ABB RAPID module: Module1.mod

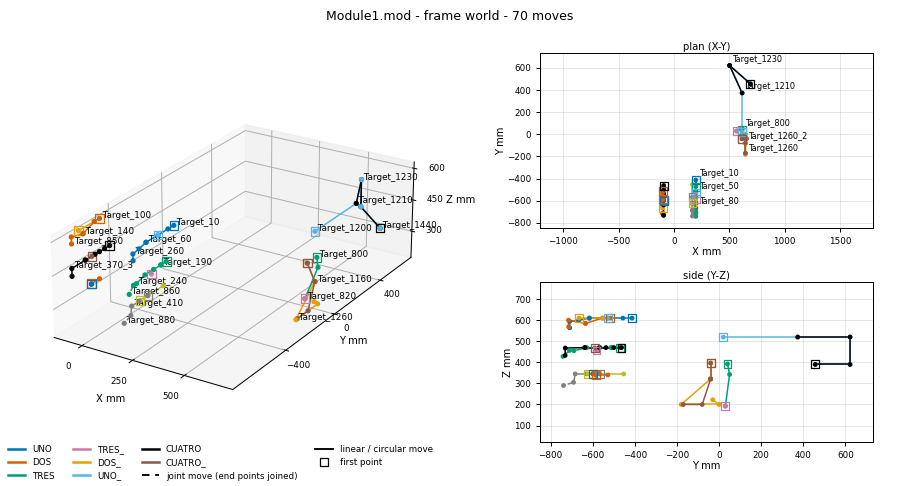
[picture p0: tool path of Module1.mod in frame world, 70 of 71 moves have a stored position in this frame; points joined in program order, loops and branches not executed]
MODULE Module1
    CONST robtarget Target_10:=[[445,309.451,360],[0,0.707106781,0.707106781,0],[-1,0,0,0],[9E+09,9E+09,9E+09,9E+09,9E+09,9E+09]];
    CONST robtarget Target_30:=[[445.000100716,265.84797315,360.000005505],[0.204070481,0.677019397,0.677019332,-0.204070573],[-1,-1,0,0],[9E+09,9E+09,9E+09,9E+09,9E+09,9E+09]];
    CONST robtarget Target_50:=[[444.999989498,193.403179869,359.99999842],[0.39678617,0.585286862,0.58528689,-0.396786191],[-1,-2,1,0],[9E+09,9E+09,9E+09,9E+09,9E+09,9E+09]];
    CONST robtarget Target_60:=[[445.000001173,106.761011861,360.000002181],[0.396786171,0.585286826,0.585286919,-0.3967862],[-1,-2,1,0],[9E+09,9E+09,9E+09,9E+09,9E+09,9E+09]];
    CONST robtarget Target_70:=[[444.999995441,106.761019962,359.999988422],[0.498060694,0.501931741,0.501931802,-0.498060778],[-1,-2,1,0],[9E+09,9E+09,9E+09,9E+09,9E+09,9E+09]];
    CONST robtarget Target_80:=[[445,56.559774308,350],[0.498058869,0.50193349,0.501933625,-0.498059004],[-1,-2,1,0],[9E+09,9E+09,9E+09,9E+09,9E+09,9E+09]];
    CONST robtarget Target_260:=[[445,13.051774308,344.078],[0.498058632,0.501933253,0.501933862,-0.498059241],[-1,-2,1,0],[9E+09,9E+09,9E+09,9E+09,9E+09,9E+09]];
    CONST robtarget Target_840:=[[445,13.283774308,314.079],[0.498058666,0.501933287,0.501933828,-0.498059207],[-1,-2,1,0],[9E+09,9E+09,9E+09,9E+09,9E+09,9E+09]];
    CONST robtarget Target_100:=[[145,206.823,360],[0,0.707106781,0.707106781,0],[-2,0,-1,0],[9E+09,9E+09,9E+09,9E+09,9E+09,9E+09]];
    CONST robtarget Target_120:=[[145.000023763,169.277992134,359.999994736],[0.208753422,0.675590111,0.675590131,-0.208753407],[-2,0,-1,0],[9E+09,9E+09,9E+09,9E+09,9E+09,9E+09]];
    CONST robtarget Target_140:=[[145,89.022774308,335],[0.308604589,0.636210034,0.636210034,-0.308604589],[-2,0,-1,0],[9E+09,9E+09,9E+09,9E+09,9E+09,9E+09]];
    CONST robtarget Target_150:=[[145,87.832774308,335],[0.308604589,0.636210034,0.636210034,-0.308604589],[-2,0,-1,0],[9E+09,9E+09,9E+09,9E+09,9E+09,9E+09]];
    CONST robtarget Target_160:=[[145,7.662774308,350.108],[0.495529584,0.504430646,0.504430801,-0.495529739],[-2,1,-2,0],[9E+09,9E+09,9E+09,9E+09,9E+09,9E+09]];
    CONST robtarget Target_850:=[[145,8.374774308,319.114],[0.495529584,0.504430646,0.504430801,-0.495529739],[-2,1,-2,0],[9E+09,9E+09,9E+09,9E+09,9E+09,9E+09]];
    CONST robtarget Target_180:=[[445,250.207,220],[0,0.707106781,0.707106781,0],[0,0,0,0],[9E+09,9E+09,9E+09,9E+09,9E+09,9E+09]];
    CONST robtarget Target_190:=[[445,210.045,220],[0,0.707106781,0.707106781,0],[-1,0,0,0],[9E+09,9E+09,9E+09,9E+09,9E+09,9E+09]];
    CONST robtarget Target_210:=[[444.999974423,210.04498181,219.999975641],[0.196714093,0.67919333,0.679193304,-0.196714112],[-1,-1,1,0],[9E+09,9E+09,9E+09,9E+09,9E+09,9E+09]];
    CONST robtarget Target_220:=[[444.999969721,157.562432775,220.000153936],[0.196714096,0.679193328,0.679193306,-0.196714111],[-1,-1,0,0],[9E+09,9E+09,9E+09,9E+09,9E+09,9E+09]];
    CONST robtarget Target_230:=[[445.000020297,94.798793532,219.999986793],[0.490571323,0.509254076,0.509254286,-0.490571233],[-1,-2,1,0],[9E+09,9E+09,9E+09,9E+09,9E+09,9E+09]];
    CONST robtarget Target_240:=[[444.99998259,33.260372465,205.010464734],[0.490571277,0.509254086,0.509254311,-0.490571243],[-1,-2,1,0],[9E+09,9E+09,9E+09,9E+09,9E+09,9E+09]];
    CONST robtarget Target_300:=[[445,12.043774308,205.998],[0.490571564,0.509254226,0.5092539,-0.490571238],[-1,-2,1,0],[9E+09,9E+09,9E+09,9E+09,9E+09,9E+09]];
    CONST robtarget Target_860:=[[445,-18.461225692,178.026],[0.49056712,0.509258507,0.509249619,-0.490575682],[-1,-2,1,0],[9E+09,9E+09,9E+09,9E+09,9E+09,9E+09]];
    CONST robtarget Target_300_2:=[[445.000076449,140.791521426,205.991567014],[0.490571145,0.509254485,0.509253958,-0.490571328],[-1,-2,1,0],[9E+09,9E+09,9E+09,9E+09,9E+09,9E+09]];
    CONST robtarget Target_170:=[[145.000002632,57.832569204,360.00000345],[0.49552756,0.504432594,0.504432809,-0.495527736],[-2,1,-2,0],[9E+09,9E+09,9E+09,9E+09,9E+09,9E+09]];
    CONST robtarget Target_120_2:=[[145.000023763,169.277992134,359.999994736],[0.208753422,0.675590111,0.675590131,-0.208753407],[-2,0,-1,0],[9E+09,9E+09,9E+09,9E+09,9E+09,9E+09]];
    CONST robtarget Target_50_2:=[[444.999989498,193.403179869,359.99999842],[0.39678617,0.585286862,0.58528689,-0.396786191],[-1,-2,1,0],[9E+09,9E+09,9E+09,9E+09,9E+09,9E+09]];
    CONST jointtarget hoome:=[[0,0,0,0,30,0],[9E+09,9E+09,9E+09,9E+09,9E+09,9E+09]];
    CONST robtarget Target_310:=[[155,259.373,220],[0,0.707106781,0.707106781,0],[-2,0,-1,0],[9E+09,9E+09,9E+09,9E+09,9E+09,9E+09]];
    CONST robtarget Target_320:=[[155,222.546,220],[0,0.707106781,0.707106781,0],[-2,0,-1,0],[9E+09,9E+09,9E+09,9E+09,9E+09,9E+09]];
    CONST robtarget Target_330:=[[154.999993427,185.47297748,219.999991899],[0.181722193,0.68335719,0.683357178,-0.181722213],[-2,0,-1,0],[9E+09,9E+09,9E+09,9E+09,9E+09,9E+09]];
    CONST robtarget Target_340:=[[155,153.836774308,220],[0.181724929,0.683356459,0.683356459,-0.181724929],[-2,0,-1,0],[9E+09,9E+09,9E+09,9E+09,9E+09,9E+09]];
    CONST robtarget Target_350:=[[155.000000465,85.426287942,219.999986272],[0.351807406,0.613377267,0.613377023,-0.351807484],[-2,1,-2,0],[9E+09,9E+09,9E+09,9E+09,9E+09,9E+09]];
    CONST robtarget Target_360:=[[155.000020231,85.426284038,219.999972166],[0.502982262,0.496999972,0.496999701,-0.502982276],[-2,1,-2,0],[9E+09,9E+09,9E+09,9E+09,9E+09,9E+09]];
    CONST robtarget Target_370_3:=[[154.117650914,-7.63964163,217.880472499],[0.502982249,0.496999966,0.496999703,-0.502982293],[-2,1,-2,0],[9E+09,9E+09,9E+09,9E+09,9E+09,9E+09]];
    CONST robtarget Target_870:=[[154.117692068,-8.05845949,182.882972826],[0.502982281,0.497000006,0.496999676,-0.502982246],[-2,1,-2,0],[9E+09,9E+09,9E+09,9E+09,9E+09,9E+09]];
    CONST robtarget Target_370_2:=[[154.117693643,132.374266615,218.205277098],[0.502982249,0.496999966,0.496999703,-0.502982293],[-2,1,-2,0],[9E+09,9E+09,9E+09,9E+09,9E+09,9E+09]];
    CONST robtarget Target_390:=[[415.000021736,155.814134714,94.99994956],[0.222483326,0.671193787,0.671193888,-0.222483337],[-1,-2,1,0],[9E+09,9E+09,9E+09,9E+09,9E+09,9E+09]];
    CONST robtarget Target_400:=[[414.999964418,93.028686316,95.000070499],[0.494470801,0.505469141,0.505468247,-0.494470854],[-1,-2,1,0],[9E+09,9E+09,9E+09,9E+09,9E+09,9E+09]];
    CONST robtarget Target_410:=[[414.999780299,39.624514396,95.000017901],[0.494470475,0.505469266,0.505467893,-0.494471414],[-1,-2,1,0],[9E+09,9E+09,9E+09,9E+09,9E+09,9E+09]];
    CONST robtarget Target_420_2:=[[415,31.615774308,55.006],[0.49447229,0.505467643,0.505467259,-0.494471906],[-1,-2,1,0],[9E+09,9E+09,9E+09,9E+09,9E+09,9E+09]];
    CONST robtarget Target_880:=[[415.000153001,-15.724115102,40.013288948],[0.49447062,0.505469365,0.505467764,-0.4944713],[-1,-2,1,0],[9E+09,9E+09,9E+09,9E+09,9E+09,9E+09]];
    CONST robtarget Target_430:=[[415.000047641,100.795599035,94.999989609],[0.494470604,0.505469297,0.505467834,-0.494471315],[-1,-2,1,0],[9E+09,9E+09,9E+09,9E+09,9E+09,9E+09]];
    CONST robtarget Target_380:=[[415,269.946,95],[0,0.707106781,0.707106781,0],[-1,0,0,0],[9E+09,9E+09,9E+09,9E+09,9E+09,9E+09]];
    CONST robtarget Target_910:=[[154.999998327,259.37294151,90.000018028],[-0.000000019,0.707106797,0.707106766,-0.000000028],[-2,0,-1,0],[9E+09,9E+09,9E+09,9E+09,9E+09,9E+09]];
    CONST robtarget Target_930:=[[155.000007698,111.881805431,90.000010525],[0.506551604,0.493361374,0.493361398,-0.506551635],[-2,1,-2,0],[9E+09,9E+09,9E+09,9E+09,9E+09,9E+09]];
    CONST robtarget Target_940:=[[155.00014811,-18.072997939,93.429168302],[0.506551657,0.493361261,0.493361508,-0.506551583],[-2,1,-2,0],[9E+09,9E+09,9E+09,9E+09,9E+09,9E+09]];
    CONST robtarget Target_950:=[[155.000223386,-19.39194722,43.446578802],[0.506551723,0.493361207,0.493361565,-0.506551516],[-2,1,-2,0],[9E+09,9E+09,9E+09,9E+09,9E+09,9E+09]];
    CONST robtarget Target_480:=[[144.999909688,137.135818312,89.9999693],[0.497141997,0.502841197,0.502842112,-0.497142208],[-2,1,-2,0],[9E+09,9E+09,9E+09,9E+09,9E+09,9E+09]];
    CONST robtarget Target_470:=[[144.999992416,137.13583322,89.999952579],[0.158251404,0.689170827,0.689170921,-0.1582514],[-2,0,-1,0],[9E+09,9E+09,9E+09,9E+09,9E+09,9E+09]];
    CONST robtarget Target_460:=[[145,194.615,90],[0,0.707106781,0.707106781,0],[-2,0,-1,0],[9E+09,9E+09,9E+09,9E+09,9E+09,9E+09]];
    CONST robtarget Target_800:=[[15.000003085,20,-7.279986715],[0.001374548,-0.707105336,0.707105556,-0.001373609],[0,-1,-1,0],[9E+09,9E+09,9E+09,9E+09,9E+09,9E+09]];
    CONST robtarget Target_810:=[[15.194319396,30.000063266,-57.279608845],[0.001374525,-0.707105304,0.707105589,-0.001373591],[0,-1,-1,0],[9E+09,9E+09,9E+09,9E+09,9E+09,9E+09]];
    CONST robtarget Target_820:=[[-34.3,9.999774308,-207.473],[0.001376059,-0.707105442,0.707105442,-0.001376059],[0,-1,-1,0],[9E+09,9E+09,9E+09,9E+09,9E+09,9E+09]];
    CONST robtarget Target_830:=[[16.049330824,30.000353686,-277.277947373],[0.001374525,-0.707105304,0.707105589,-0.001373591],[0,-1,-1,0],[9E+09,9E+09,9E+09,9E+09,9E+09,9E+09]];
    CONST robtarget Target_960:=[[15,-60.000225692,-3.34],[0.422618262,0,0.906307787,0],[-1,0,-1,0],[9E+09,9E+09,9E+09,9E+09,9E+09,9E+09]];
    CONST robtarget Target_980:=[[15.000003989,-60.000225846,-65.005610701],[0.698090332,-0.000000037,0.716009699,-0.000000028],[-1,1,-2,0],[9E+09,9E+09,9E+09,9E+09,9E+09,9E+09]];
    CONST robtarget Target_990:=[[64.983949086,-84.888859881,-188.758694739],[0.698090343,-0.000000088,0.716009688,0.00000008],[-1,1,-2,0],[9E+09,9E+09,9E+09,9E+09,9E+09,9E+09]];
    CONST robtarget Target_1000:=[[64.983940199,-84.888856272,-260.223415545],[0.698090318,-0.000000083,0.716009712,0.000000092],[-1,1,-2,0],[9E+09,9E+09,9E+09,9E+09,9E+09,9E+09]];
    CONST robtarget Target_1010:=[[64.983925895,-54.888697083,-260.223308264],[0.698090428,-0.000000715,0.716009604,0.000000241],[-1,1,-2,0],[9E+09,9E+09,9E+09,9E+09,9E+09,9E+09]];
    CONST robtarget Target_1020:=[[67.517875393,-54.888638408,-160.255409875],[0.698090412,-0.000000696,0.716009621,0.000000195],[-1,1,-2,0],[9E+09,9E+09,9E+09,9E+09,9E+09,9E+09]];
    CONST robtarget Target_1030:=[[1115.000003258,-650.827226308,222.202998223],[0.342020143,0,0.939692621,0],[0,-1,0,0],[9E+09,9E+09,9E+09,9E+09,9E+09,9E+09]];
    CONST robtarget Target_1040:=[[1115.000009669,-650.827230544,392.898398622],[0.683149215,-0.147345411,0.700684713,0.143657274],[-1,1,-2,0],[9E+09,9E+09,9E+09,9E+09,9E+09,9E+09]];
    CONST robtarget Target_1050:=[[1115.000011784,-558.507726654,392.898390868],[0.683149204,-0.14734549,0.700684704,0.143657288],[0,1,-2,0],[9E+09,9E+09,9E+09,9E+09,9E+09,9E+09]];
    CONST robtarget Target_1060:=[[1115.000006212,-451.354920054,392.898384166],[0.683149189,-0.14734552,0.700684714,0.143657286],[0,1,-2,0],[9E+09,9E+09,9E+09,9E+09,9E+09,9E+09]];
    CONST robtarget Target_1080:=[[998.889389949,-391.005407979,392.898398132],[0.683149203,-0.147345556,0.700684696,0.143657271],[0,2,-3,0],[9E+09,9E+09,9E+09,9E+09,9E+09,9E+09]];
    CONST robtarget Target_1090:=[[865.105301275,-168.564929633,392.898396083],[0.616538883,-0.335834912,0.632364278,0.327429593],[0,1,-2,0],[9E+09,9E+09,9E+09,9E+09,9E+09,9E+09]];
    CONST robtarget Target_1100:=[[878.271514464,-30.097814532,392.898393764],[0.616538885,-0.335835049,0.632364231,0.327429538],[0,2,-3,0],[9E+09,9E+09,9E+09,9E+09,9E+09,9E+09]];
    CONST robtarget Target_1110:=[[878.271453157,-30.097779623,331.594271959],[0.616538889,-0.33583503,0.632364227,0.327429558],[0,2,-3,0],[9E+09,9E+09,9E+09,9E+09,9E+09,9E+09]];
    CONST robtarget Target_1120:=[[927.980685621,-63.698381666,331.594348136],[0.6165389,-0.335835004,0.632364219,0.32742958],[0,1,-2,0],[9E+09,9E+09,9E+09,9E+09,9E+09,9E+09]];
    CONST robtarget Target_1130:=[[929.115831572,-62.018793499,411.568574487],[0.616538876,-0.335835031,0.63236422,0.327429593],[0,1,-2,0],[9E+09,9E+09,9E+09,9E+09,9E+09,9E+09]];
    CONST robtarget Target_1140:=[[155.00004953,123.02170152,95.65965675],[0.494470878,0.50546913,0.505468146,-0.494470891],[-2,1,-2,0],[9E+09,9E+09,9E+09,9E+09,9E+09,9E+09]];
    CONST robtarget Target_1190:=[[45,-50.000225692,-177.596],[0.574790179,-0.270574227,0.743396577,-0.209206516],[-1,0,-1,0],[9E+09,9E+09,9E+09,9E+09,9E+09,9E+09]];
    CONST robtarget Target_1170:=[[15,-100.000225692,-269.732],[0.342020143,0,0.939692621,0],[-1,0,-1,0],[9E+09,9E+09,9E+09,9E+09,9E+09,9E+09]];
    CONST robtarget Target_1180:=[[45,-50.000225692,-271.262],[0.611678933,0,0.791106114,0],[-1,0,-1,0],[9E+09,9E+09,9E+09,9E+09,9E+09,9E+09]];
    CONST robtarget Target_1260:=[[45,-200.000225692,-200],[0.602385883,-0.137375677,0.779087162,-0.106218474],[-1,1,-2,0],[9E+09,9E+09,9E+09,9E+09,9E+09,9E+09]];
    CONST robtarget Target_1150:=[[15,-60.000225692,-24.284],[0.173648178,0,0.984807753,0],[-1,0,-1,0],[9E+09,9E+09,9E+09,9E+09,9E+09,9E+09]];
    CONST robtarget Target_1160:=[[52.587704822,-60.000225692,-78.767194242],[0.173648178,0,0.984807753,0],[-1,0,-1,0],[9E+09,9E+09,9E+09,9E+09,9E+09,9E+09]];
    CONST robtarget Target_1250:=[[1167.584,-194.402225692,410],[0.31160272,-0.387399417,0.856121436,0.141001857],[0,0,-1,0],[9E+09,9E+09,9E+09,9E+09,9E+09,9E+09]];
    CONST robtarget Target_1240:=[[1002.320747823,-49.18417527,390.000000069],[0.341036269,-0.656847149,0.671992582,0.025924035],[0,0,-1,0],[9E+09,9E+09,9E+09,9E+09,9E+09,9E+09]];
    CONST robtarget Target_1230:=[[1002.32107139,-49.183439733,519.999883014],[0.311602972,-0.387398085,0.856122024,0.141001388],[0,0,-1,0],[9E+09,9E+09,9E+09,9E+09,9E+09,9E+09]];
    CONST robtarget Target_1210:=[[1115.000004816,-297.587934649,519.999950749],[0.342020175,0.00000003,0.939692609,-0.000000022],[0,-1,0,0],[9E+09,9E+09,9E+09,9E+09,9E+09,9E+09]];
    CONST robtarget Target_1200:=[[1115,-650.827225692,520],[0.342020143,0,0.939692621,0],[0,-1,0,0],[9E+09,9E+09,9E+09,9E+09,9E+09,9E+09]];
    CONST robtarget Target_1280:=[[52.587712308,-60.000227715,-78.767220897],[0.440689623,-0.000000022,0.897659543,-0.000000013],[-1,0,-1,0],[9E+09,9E+09,9E+09,9E+09,9E+09,9E+09]];
    CONST robtarget Target_1440:=[[1190.119504813,-214.204262911,389.999988496],[0.341036269,-0.656847149,0.671992582,0.025924035],[0,0,-1,0],[9E+09,9E+09,9E+09,9E+09,9E+09,9E+09]];
    CONST robtarget Target_1260_2:=[[45,-100.000225692,-200],[0.554368788,-0.334338154,0.716984512,-0.258508131],[-1,1,-2,0],[9E+09,9E+09,9E+09,9E+09,9E+09,9E+09]];
    CONST robtarget Target_1460:=[[45.000159369,-190.000214557,-199.999516221],[0.611679058,-0.000002498,0.791106017,-0.000001528],[-1,1,-2,0],[9E+09,9E+09,9E+09,9E+09,9E+09,9E+09]];

PROC main()
    WaitDI DI_01,1;  // Espera hasta que la entrada DI_01 sea igual a 1.
    SETDO DO_03,1;   // Establece la salida DO_03 en 1.
    homee;           // Mueve el robot a la posición de origen (home).
    BaldeR;          // Toma el balde de la banda.
    homee;           // Vuelve a la posición de origen.
    BaldeR1;         // posiciona el balde.
    homee;           // Vuelve a la posición de origen.
    UNO;             // Toma ficha.
    SETDO DO_01,0;   // Establece la salida DO_01 en 0.
    SETDO DO_02,1;   // Establece la salida DO_02 en 1.
    WaitTime 3;      // Espera durante 3 segundos.
    UNO_;            // Retira la ficha.
    homee;           // Vuelve a la posición de origen.
    dejarFichas;     // Deja la ficha en el balde.
    WaitTime 3;      // Espera durante 3 segundos.
    SETDO DO_01,1;   // Establece la salida DO_01 en 1.
    SETDO DO_02,0;   // Establece la salida DO_02 en 0.
    WaitTime 2;      // Espera durante 2 segundos.
    homee;           // Vuelve a la posición de origen.

    DOS;             // Toma ficha.
    SETDO DO_01,0;   // Establece la salida DO_01 en 0.
    SETDO DO_02,1;   // Establece la salida DO_02 en 1.
    WaitTime 3;      // Espera durante 3 segundos.
    DOS_;            // Retira la ficha.
    homee;           // Vuelve a la posición de origen.
    dejarFichas;     // Deja la ficha en el balde.
    WaitTime 3;      // Espera durante 3 segundos.
    SETDO DO_01,1;   // Establece la salida DO_01 en 1.
    SETDO DO_02,0;   // Establece la salida DO_02 en 0.
    WaitTime 2;      // Espera durante 2 segundos.
    homee;           // Vuelve a la posición de origen.

    TRES;            // toma ficha.
    SETDO DO_01,0;   // Establece la salida DO_01 en 0.
    SETDO DO_02,1;   // Establece la salida DO_02 en 1.
    WaitTime 3;      // Espera durante 3 segundos.
    TRES_;           // Retira la ficha.
    homee;           // Vuelve a la posición de origen.
    dejarFichas;     // Deja la ficha en el balde.
    WaitTime 3;      // Espera durante 3 segundos.
    SETDO DO_01,1;   // Establece la salida DO_01 en 1.
    SETDO DO_02,0;   // Establece la salida DO_02 en 0.
    WaitTime 2;      // Espera durante 2 segundos.
    homee;           // Vuelve a la posición de origen.

    Balde1;          // Toma el balde.
    homee;           // Vuelve a la posición de origen.
    Balde2;          // Deja el balde en la banda.
    homee;           // Vuelve a la posición de origen.

    SETDO DO_03,0;   // Establece la salida DO_03 en 0.
ENDPROC


    PROC UNO()
        MoveL Target_10,v500,z100,HerramientaP\WObj:=Estante;
        MoveL Target_30,v500,z100,HerramientaP\WObj:=Estante;
        MoveL Target_50,v500,z100,HerramientaP\WObj:=Estante;
        MoveL Target_60,v500,z100,HerramientaP\WObj:=Estante;
        MoveL Target_70,v500,z100,HerramientaP\WObj:=Estante;
        MoveL Target_80,v500,z100,HerramientaP\WObj:=Estante;
        MoveL Target_260,v500,z100,HerramientaP\WObj:=Estante;
        MoveJ Target_840,v1000,z100,HerramientaP\WObj:=Estante;
    ENDPROC
    PROC DOS()
        MoveL Target_100,v300,z100,HerramientaP\WObj:=Estante;
        MoveL Target_120,v300,z100,HerramientaP\WObj:=Estante;
        MoveL Target_140,v300,z100,HerramientaP\WObj:=Estante;
        MoveL Target_150,v300,z100,HerramientaP\WObj:=Estante;
        MoveL Target_160,v300,z100,HerramientaP\WObj:=Estante;
        MoveJ Target_850,v1000,z100,HerramientaP\WObj:=Estante;
    ENDPROC
    PROC TRES()
        MoveL Target_180,v500,z100,HerramientaP\WObj:=Estante;
        MoveL Target_190,v500,z100,HerramientaP\WObj:=Estante;
        MoveL Target_210,v500,z100,HerramientaP\WObj:=Estante;
        MoveL Target_220,v500,z100,HerramientaP\WObj:=Estante;
        MoveL Target_230,v500,z100,HerramientaP\WObj:=Estante;
        MoveL Target_240,v500,z100,HerramientaP\WObj:=Estante;
        MoveL Target_300,v500,z100,HerramientaP\WObj:=Estante;
        MoveJ Target_860,v1000,z100,HerramientaP\WObj:=Estante;
    ENDPROC
    PROC TRES_()
        MoveL Target_300_2,v300,z100,HerramientaP\WObj:=Estante;
    ENDPROC
    PROC DOS_()
        MoveL Target_170,v300,z100,HerramientaP\WObj:=Estante;
        MoveL Target_120_2,v300,z100,HerramientaP\WObj:=Estante;
    ENDPROC
    PROC UNO_()
        MoveL Target_50_2,v500,z100,HerramientaP\WObj:=Estante;
    ENDPROC
    PROC homee()
        MoveAbsJ hoome,v1000,z100,HerramientaP\WObj:=Estante;
    ENDPROC
    PROC CUATRO()
        MoveL Target_310,v300,z100,HerramientaP\WObj:=Estante;
        MoveL Target_320,v300,z100,HerramientaP\WObj:=Estante;
        MoveL Target_330,v300,z100,HerramientaP\WObj:=Estante;
        MoveL Target_340,v300,z100,HerramientaP\WObj:=Estante;
        MoveL Target_350,v300,z100,HerramientaP\WObj:=Estante;
        MoveL Target_360,v300,z100,HerramientaP\WObj:=Estante;
        MoveL Target_370_3,v300,z100,HerramientaP\WObj:=Estante;
        MoveJ Target_870,v1000,z100,HerramientaP\WObj:=Estante;
    ENDPROC
    PROC CUATRO_()
        MoveL Target_370_2,v300,z100,HerramientaP\WObj:=Estante;
    ENDPROC
    PROC CINCO()
        MoveL Target_390,v300,z100,HerramientaP\WObj:=Estante;
        MoveL Target_400,v300,z100,HerramientaP\WObj:=Estante;
        MoveL Target_410,v300,z100,HerramientaP\WObj:=Estante;
        MoveL Target_420_2,v300,z100,HerramientaP\WObj:=Estante;
        MoveJ Target_880,v1000,z100,HerramientaP\WObj:=Estante;
    ENDPROC
    PROC CINCO_()
        MoveL Target_430,v300,z100,HerramientaP\WObj:=Estante;
        MoveL Target_380,v300,z100,HerramientaP\WObj:=Estante;
    ENDPROC
    PROC SEIS()
        MoveJ Target_1140,v300,z100,HerramientaP\WObj:=Estante;
    ENDPROC
    PROC SEIS_()
        MoveL Target_480,v300,z100,HerramientaP\WObj:=Estante;
        MoveL Target_470,v300,z100,HerramientaP\WObj:=Estante;
        MoveL Target_460,v300,z100,HerramientaP\WObj:=Estante;
    ENDPROC
    PROC dejarFichas()
        MoveL Target_800,v200,z100,HerramientaP\WObj:=Balde;
        MoveL Target_810,v200,z100,HerramientaP\WObj:=Balde;
        MoveL Target_820,v200,z100,HerramientaP\WObj:=Balde;
    ENDPROC
    PROC dejarFichas_()
        MoveJ Target_820,v1000,z100,HerramientaP\WObj:=Balde;
    ENDPROC
    PROC Balde1()
        MoveL Target_960,v300,z100,HerramientaP\WObj:=Balde;
        MoveL Target_1160,v300,z100,HerramientaP\WObj:=Balde;
        MoveL Target_1280,v300,z100,HerramientaP\WObj:=Balde;
        MoveL Target_1260,v300,z100,HerramientaP\WObj:=Balde;
        MoveL [[45,-20.000225692,-200],[0.574789716,-0.270576578,0.74339566,-0.209208006],[-1,0,-1,0],[9E+09,9E+09,9E+09,9E+09,9E+09,9E+09]],v300,z100,HerramientaP\WObj:=Balde;
        MoveL Target_1190,v300,z100,HerramientaP\WObj:=Balde;
    ENDPROC
    PROC Balde2()
        MoveL Target_1200,v300,z100,HerramientaP\WObj:=Banda;
        MoveL Target_1210,v300,z100,HerramientaP\WObj:=Banda;
        MoveL Target_1230,v100,z100,HerramientaP\WObj:=Banda;
        MoveL Target_1240,v100,z100,HerramientaP\WObj:=Banda;
        MoveL Target_1440,v100,z100,HerramientaP\WObj:=Banda;
    ENDPROC
    PROC BaldeR()
        MoveL Target_1440,v300,z100,HerramientaP\WObj:=Banda;
        MoveL Target_1240,v300,z100,HerramientaP\WObj:=Banda;
        MoveL Target_1230,v300,z100,HerramientaP\WObj:=Banda;
        MoveL Target_1210,v100,z100,HerramientaP\WObj:=Banda;

    ENDPROC
    PROC BaldeR1()
        MoveL Target_960,v300,z100,HerramientaP\WObj:=Balde;
        MoveL Target_1160,v300,z100,HerramientaP\WObj:=Balde;
        MoveL Target_1280,v300,z100,HerramientaP\WObj:=Balde;
        MoveL Target_1260_2,v300,z100,HerramientaP\WObj:=Balde;
        MoveL Target_1460,v300,z100,HerramientaP\WObj:=Balde;
    ENDPROC
ENDMODULE
